FUNCTION_BLOCK FB_ThNTZ_Ablaufsteuerung
VAR_IN_OUT
	Zustand				: ST_ThNTZ_Zustand;
	Stellwert			: ST_ThNTZ_Stellwert;
	Steuerung			: ST_ThNTZ_Steuerung;
END_VAR
VAR_INPUT
END_VAR
VAR_OUTPUT
END_VAR
VAR
END_VAR

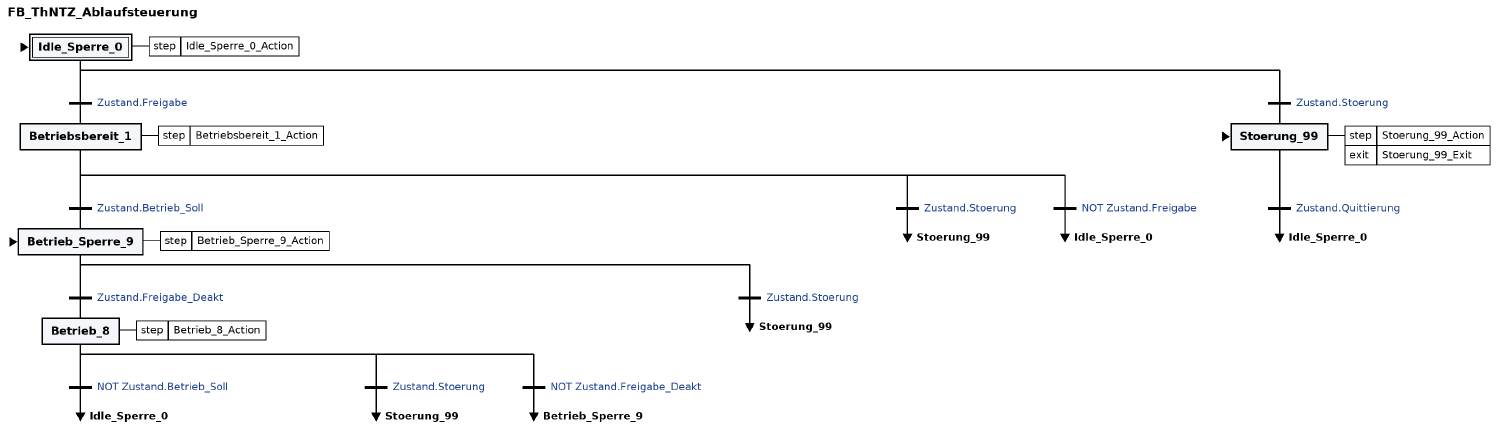
INITIAL_STEP Idle_Sperre_0:
    Idle_Sperre_0_Action(N);  // step action
END_STEP
TRANSITION FROM Idle_Sperre_0 TO Betriebsbereit_1
    := Zustand.Freigabe;
END_TRANSITION
TRANSITION FROM Idle_Sperre_0 TO Stoerung_99
    := Zustand.Stoerung;
END_TRANSITION
STEP Stoerung_99:
    Stoerung_99_Action(N);  // step action
    Stoerung_99_Exit(P0);  // exit action
END_STEP
TRANSITION FROM Stoerung_99 TO Idle_Sperre_0
    := Zustand.Quittierung;
END_TRANSITION
STEP Betriebsbereit_1:
    Betriebsbereit_1_Action(N);  // step action
END_STEP
TRANSITION FROM Betriebsbereit_1 TO Betrieb_Sperre_9
    := Zustand.Betrieb_Soll;
END_TRANSITION
TRANSITION FROM Betriebsbereit_1 TO Stoerung_99
    := Zustand.Stoerung;
END_TRANSITION
TRANSITION FROM Betriebsbereit_1 TO Idle_Sperre_0
    := NOT Zustand.Freigabe;
END_TRANSITION
STEP Betrieb_Sperre_9:
    Betrieb_Sperre_9_Action(N);  // step action
END_STEP
TRANSITION FROM Betrieb_Sperre_9 TO Betrieb_8
    := Zustand.Freigabe_Deakt;
END_TRANSITION
TRANSITION FROM Betrieb_Sperre_9 TO Stoerung_99
    := Zustand.Stoerung;
END_TRANSITION
STEP Betrieb_8:
    Betrieb_8_Action(N);  // step action
END_STEP
TRANSITION FROM Betrieb_8 TO Idle_Sperre_0
    := NOT Zustand.Betrieb_Soll;
END_TRANSITION
TRANSITION FROM Betrieb_8 TO Stoerung_99
    := Zustand.Stoerung;
END_TRANSITION
TRANSITION FROM Betrieb_8 TO Betrieb_Sperre_9
    := NOT Zustand.Freigabe_Deakt;
END_TRANSITION

ACTION Betrieb_8_Action:
(* Stellwert setzen *)
Stellwert.Betrieb				:= TRUE;
Zustand.Betrieb				:= TRUE;

(* Zustand setzen *)
Zustand.Status				:= E_ThNTZ_Zustand_Status_Betrieb;
END_ACTION

ACTION Betrieb_Sperre_9_Action:
(* Stellwert setzen *)
Stellwert.Betrieb				:= TRUE;
Zustand.Betrieb				:= TRUE;

(* Zustand setzen *)
Zustand.Status				:= E_ThNTZ_Zustand_Status_Betrieb_Sperre;
END_ACTION

ACTION Betriebsbereit_1_Action:
(* Stellwert setzen *)
Stellwert.Betrieb		:= FALSE;
Zustand.Betrieb		:= FALSE;

(* Zustand setzen *)
Zustand.Status			:= E_ThNTZ_Zustand_Status_Betriebsbereit;
END_ACTION

ACTION Idle_Sperre_0_Action:
(* Stellwert setzen *)
Stellwert.Betrieb		:= FALSE;
Zustand.Betrieb		:= FALSE;

(* Zustand setzen *)
Zustand.Status				:= E_ThNTZ_Zustand_Status_Idle_Sperre;

(* Quittierungszustand auf False setzen, damit das System bei einer erneuten Störung nicht direkt wieder angeschaltet wird *)
Steuerung.Quittierung	:= FALSE;
END_ACTION

ACTION Stoerung_99_Action:
(* Stellwert setzen *)
Stellwert.Betrieb			:= FALSE;
Zustand.Betrieb			:= FALSE;

(* Zustand setzen *)
Zustand.Stoerung			:= TRUE;
Zustand.Status			:= E_ThNTZ_Zustand_Status_Stoerung;
END_ACTION

ACTION Stoerung_99_Exit:
Zustand.Stoerung	:= FALSE;
END_ACTION

END_FUNCTION_BLOCK

(* stored: Version 1.1.0.1, ProductVersion 3.1.4024.9
   POU FB_ThNTZ_Ablaufsteuerung: Id {9b72176d-31a4-48ee-b59b-1c173baf22fd}, SpecialFunc None
   Action Betrieb_8_Action: Id {4b3eccf6-ea2b-4385-b577-d4337e2544ac}
   Action Betrieb_Sperre_9_Action: Id {6b688bb6-c72f-4e00-baa2-337b22e952a5}
   Action Betriebsbereit_1_Action: Id {323e29da-57eb-429a-bcb4-4c970175ee8a}
   Action Idle_Sperre_0_Action: Id {b8bab1d3-9925-47c2-8c5e-167095a2fbb6}
   Action Stoerung_99_Action: Id {952f8c1b-868c-496b-b5f1-9bdf210075ac}
   Action Stoerung_99_Exit: Id {1ff0c11b-a938-422b-b364-508be066d44f} *)
